// TIA Portal V19 export
TYPE "LUC_typeStates"
// stored: Access Published
   STRUCT
      current : DInt;   // Current unit state
      clearing : Bool;   // The unit state "Clearing" is active
      stopped : Bool;   // The unit state "Stopped" is active
      starting : Bool;   // The unit state "Starting" is active
      idle : Bool;   // The unit state "Idle" is active
      suspended : Bool;   // The unit state "Suspended" is active
      execute : Bool;   // The unit state "Execute" is active
      stopping : Bool;   // The unit state "Stopping" is active
      aborting : Bool;   // The unit state "Aborting" is active
      aborted : Bool;   // The unit state "Aborted" is active
      holding : Bool;   // The unit state "Holding" is active
      held : Bool;   // The unit state "Held" is active
      unholding : Bool;   // The unit state "Unholding" is active
      suspending : Bool;   // The unit state "Suspending" is active
      unsuspending : Bool;   // The unit state "Unsuspending" is active
      resetting : Bool;   // The unit state "Resetting" is active
      completing : Bool;   // The unit state "Completing" is active
      complete : Bool;   // The unit state "Complete" is active
   END_STRUCT;
END_TYPE
